TYPE ST_KNX_DPT_B2 :
STRUCT
	bBit1			: BOOL;
	bBit2			: BOOL;
END_STRUCT
END_TYPE

(* stored: Version 1.1.0.1
   DUT ST_KNX_DPT_B2: Id {f7cc3e67-ca70-4c7b-9e0d-24f7eb1fb506} *)
